(* PLC project pc, TNI-Software ControlBuild 4.00 *)
(* stored: creationDateTime 2018-09-17T17:24:47-01:00 *)

PROGRAM tapis_conv.pc
  VAR_INPUT  (* CB.group=Retour_PO CB.kind=inputVars *)
    Fin_Convoyage : BOOL := false;
  END_VAR
  VAR_INPUT  (* CB.group=Retour_Utilisateur CB.kind=inputVars *)
    Chargement : BOOL := false;
    Dechargement : BOOL := false;
  END_VAR
  VAR_OUTPUT  (* CB.group=Commande_PO CB.kind=outputVars *)
    Marche : BOOL := false;
  END_VAR

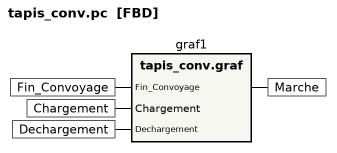
(* FBD diagram, written out as Structured Text *)
graf1(Fin_Convoyage := Fin_Convoyage, Chargement := Chargement, Dechargement := Dechargement);
Marche := graf1.Marche;
END_PROGRAM
